FUNCTION_BLOCK FB_Sealer EXTENDS FB_PackML_BaseModule
VAR
    // Sub module definitions here

    // List of sub modules
    ipSubModules_Init : ARRAY[1..Parameters_PackML_Base.MAX_NO_OF_SUBMODULES] OF I_PackML_BaseModule := [];

    // Component definitions here
    SealerAxis : FB_Component_BasicAxis := (Name := 'Axis');
    SealBar    : FB_SealBar             := (Name := 'Heat Bar');

    //Alarms for this module
    SealerAlarms : ARRAY[1..SEALER_ALARM_COUNT] OF FB_TcAlarm;

    //Data for recipe
    Recipe : ST_SealerRecipe;

    (*//Parameters from PackTags for module
    _Param  : ARRAY[1..10] OF ST_Descriptor2;*)
    _Report : ARRAY[1..10] OF ST_Descriptor2;

    //HMI Control for EM
    fbControlSourceHMI : FB_ControlSource_HMI;
END_VAR

VAR CONSTANT

    // Report parameters 
    FAULTID  : INT := 1; //Fault number 
    CURRTEMP : INT := 2; // current temperature of the sealing bar 
    CURRPOS  : INT := 3; // current position of the sealing bar  

    //Alarms
    SEALER_ALARM_COUNT : INT := 6;
END_VAR

//Simulation variables for messaging
VAR
    ErrorInput      : BOOL;
    WarnInput       : BOOL;
    InfoInput       : BOOL;
    TempFeedbackBad : BOOL;
END_VAR

METHOD PROTECTED Aborting
VAR_INPUT
END_VAR
CASE SequenceState OF
    0:
        NoStateTasksToComplete := FALSE;
        SequenceState          := SequenceState + 10;
    10:
        SealBar.Heat := FALSE;
        SealerAxis.Stop();
        IF SealerAxis.Stopped THEN
            SequenceState := SequenceState + 10;
        END_IF
    20:
        // Disable here
        SealerAxis.Disable();

        // Check not enabled here
        IF NOT SealerAxis.Enabled THEN
            SequenceState := SequenceState + 10;
        END_IF
    30:
        StateTasksComplete := TRUE;
END_CASE

SUPER^.Aborting();
END_METHOD

PROPERTY Acceleration : LREAL
SET
Recipe.Axis.Acceleration := Acceleration;
END_SET
END_PROPERTY

METHOD PROTECTED Clearing
VAR_INPUT
END_VAR
CASE SequenceState OF
    0:
        NoStateTasksToComplete := FALSE;
        SequenceState          := SequenceState + 10;
    10:
        // Enable here
        SealerAxis.Enable();

        // Check enabled here
        IF SealerAxis.Enabled THEN
            SequenceState := SequenceState + 10;
        END_IF
    20:
        StateTasksComplete := TRUE;
END_CASE

SUPER^.Clearing();
END_METHOD

PROPERTY ClosedPos : LREAL
GET
ClosedPos := Recipe.ClosedPosition;
END_GET
SET
Recipe.ClosedPosition := ClosedPos;
END_SET
END_PROPERTY

METHOD PROTECTED CreateEvents
VAR_INPUT
END_VAR
// Add your event creation here
F_CreateAllEventsInClass(Alarms     := SealerAlarms,
                         ClassSize  := SIZEOF(TC_EVENTS.Sealer),
                         pInitEvent := ADR(TC_EVENTS.Sealer.InitReferenceEvent),
                         Prefix     := Name);

// Super call to base
SUPER^.CreateEvents();
END_METHOD

METHOD CyclicLogic
VAR_INPUT
END_VAR

VAR
    LowLimit  : STRING;
    HighLimit : STRING;
END_VAR
IF NOT _InitComplete THEN
    _InitComplete := Initialize();
    RETURN;
END_IF

SUPER^.CyclicLogic();
CyclicLogic_Simulation();

//HMI control for EM
fbControlSourceHMI.CyclicLogic();

//Set the current alarm severity for this module
_CurrentAlarmSeverity   := F_GetMaxSeverityRaised(Alarms := SealerAlarms, CurrentSeverity := _CurrentAlarmSeverity);
_Report[CURRTEMP].Value := SealBar.ActualTemperature;
_Report[CURRPOS].Value  := SealerAxis.ActualPosition;

//Monitor seal bar temp
IF NOT SealBar.InTempRange AND NOT SealerAlarms[E_Sealer.TemeratureOutOfRange].bRaised THEN
    LowLimit  := TO_STRING(SealBar.SetTemperature - 1);
    HighLimit := TO_STRING(SealBar.SetTemperature + 1);
    RaiseAlarm2Args(SealerAlarms[E_Sealer.TemeratureOutOfRange], LowLimit, HighLimit);
ELSIF SealBar.InTempRange AND SealerAlarms[E_Sealer.TemeratureOutOfRange].bRaised THEN
    SealerAlarms[E_Sealer.TemeratureOutOfRange].Clear(0, 0);
END_IF
END_METHOD

METHOD CyclicLogic_Simulation
VAR_INPUT
END_VAR

VAR_INST
END_VAR
(*	
This is just for testing. Real hardware can be setup in other places
Here the alarms will raise and clear on its own if the input changes	
*)

//Generic Alarms for Testing
IF ErrorInput AND NOT SealerAlarms[E_Sealer.AlarmMessage].bRaised THEN
    RaiseAlarm2Args(SealerAlarms[E_Sealer.AlarmMessage], '', '');
ELSIF NOT ErrorInput AND SealerAlarms[E_Sealer.AlarmMessage].bRaised THEN
    SealerAlarms[E_Sealer.AlarmMessage].Clear(0, 0);
END_IF

IF WarnInput AND NOT SealerAlarms[E_Sealer.WarnMessage].bRaised THEN
    RaiseAlarm2Args(SealerAlarms[E_Sealer.WarnMessage], '', '');
ELSIF NOT WarnInput AND SealerAlarms[E_Sealer.WarnMessage].bRaised THEN
    SealerAlarms[E_Sealer.WarnMessage].Clear(0, 0);
END_IF

IF InfoInput AND NOT SealerAlarms[E_Sealer.InfoMessage].bRaised THEN
    RaiseAlarm2Args(SealerAlarms[E_Sealer.InfoMessage], '', '');
ELSIF NOT InfoInput AND SealerAlarms[E_Sealer.InfoMessage].bRaised THEN
    SealerAlarms[E_Sealer.InfoMessage].Clear(0, 0);
END_IF

// Only here for simulating alarm
IF TempFeedbackBad AND NOT SealerAlarms[E_Sealer.FeedbackError].bRaised THEN
    RaiseAlarm2Args(SealerAlarms[E_Sealer.FeedbackError], '', '');
ELSIF NOT TempFeedbackBad AND SealerAlarms[E_Sealer.FeedbackError].bRaised THEN
    SealerAlarms[E_Sealer.FeedbackError].Clear(0, 0);
END_IF
END_METHOD

METHOD PROTECTED Execute
VAR_INPUT
END_VAR

VAR_INST
    dwellTime : TON;
END_VAR
CASE _CurrentMode OF
    //=================================PRODUCTION MODE==================================
    E_PMLUnitMode.ePMLUnitMode_Production:
        CASE SequenceState OF
            0:
                IF SealerAxis.InPosition AND NOT SealerAxis.Busy THEN
                    /// SealerAxis needs to do reporting here?? no tags in the components for PackML so should be done with this module
                    dwellTime(IN := TRUE, PT := LREAL_TO_TIME(Recipe.SealTime));
                    SequenceState := SequenceState + 10;
                END_IF
            10:
                IF dwellTime.Q THEN
                    dwellTime(IN := FALSE);
                    SealerAxis.Velocity     := Recipe.Axis.Velocity;    
                    SealerAxis.Acceleration := Recipe.Axis.Acceleration;
                    SealerAxis.MoveAbsolute(Position := Recipe.OpenPosition, FALSE);
                    SequenceState := SequenceState + 10;
                END_IF
            20:
                IF SealerAxis.InPosition AND NOT SealerAxis.Busy THEN
                    ///SealerAxis report position?
                    StateComplete();
                END_IF
        END_CASE

        dwellTime();

    //=================================MAINTENANCE & MANUAL MODE==================================		
    E_PMLUnitMode.ePMLUnitMode_Maintenance, E_PMLUnitMode.ePMLUnitMode_Manual:
        ;
END_CASE
END_METHOD

PROPERTY Heat : BOOL
GET
Heat := SealBar.Heat;
END_GET
SET
SealBar.Heat := Heat;
END_SET
END_PROPERTY

//! @summary Basic module initialization logic
METHOD PROTECTED Initialize : BOOL;
VAR
    i                        : UDINT;
    varInfo                  : __SYSTEM.VAR_INFO;
    AllSubUnitsInitialized   : BOOL := TRUE;
    AllComponentsInitialized : BOOL := TRUE;
END_VAR

//! @description This method is called by <c>CyclicLogic()</c> as required
Initialize := FALSE;
CASE DescendantSequenceState OF
    0:
		RegisterComponent(SealerAxis);
		RegisterComponent(SealBar);
		
        _LogModeChanges         := FALSE;
        _LogStateChanges        := FALSE;
        DescendantSequenceState := DescendantSequenceState + 10;
    10:
        //Setup Custom modes here

        (*CustomModes(eMode                          :=,
                    sName                          :=,
                    bDisableClearing               :=,
                    bDisableStarting               :=,
                    bDisableSuspended              :=,
                    bDisableStopping               :=,
                    bDisableAborting               :=,
                    bDisableHolding                :=,
                    bDisableHeld                   :=,
                    bDisableUnholding              :=,
                    bDisableSuspending             :=,
                    bDisableUnsuspending           :=,
                    bDisableResetting              :=,
                    bDisableIdle                   :=,
                    bDisableCompleting             :=,
                    bDisableComplete               :=,
                    bEnableUnitModeChangeStopped   :=,
                    bEnableUnitModeChangeIdle      :=,
                    bEnableUnitModeChangeSuspended :=,
                    bEnableUnitModeChangeExecute   :=,
                    bEnableUnitModeChangeAborted   :=,
                    bEnableUnitModeChangeHeld      :=,
                    bEnableUnitModeChangeComplete  :=,
                    bError                         =>,
                    nErrorId                       =>);*)
        DescendantSequenceState := DescendantSequenceState + 10;
    20:
        //Copy Mode names
        FOR i := 1 TO 3 DO
            ModeNames[i] := F_UnitModeToString(UDINT_TO_DINT(i));
        END_FOR

        Initialize_TagData();
		RegisterExternalController(Controller := fbControlSourceHMI);
		fbControlSourceHMI.CyclicLogic();
        DescendantSequenceState := DescendantSequenceState + 10;
    30:
        //Call the Super
        IF SUPER^.Initialize() THEN
            DescendantSequenceState := DescendantSequenceState + 10;
        END_IF
    40:
        Initialize := TRUE;
END_CASE
END_METHOD

METHOD Initialize_TagData
VAR_INPUT
END_VAR
//Reports
_Report[FAULTID].ID    := TO_DINT(2 * 10 + 1);
_Report[FAULTID].Name  := 'Fault';
_Report[FAULTID].Unit  := '';
_Report[CURRPOS].ID    := TO_DINT(2 * 10 + 2);
_Report[CURRPOS].Name  := 'Seal Pos';
_Report[CURRPOS].Unit  := 'deg';
_Report[CURRTEMP].ID   := TO_DINT(2 * 10 + 3);
_Report[CURRTEMP].Name := 'Seal Temp';
_Report[CURRTEMP].Unit := 'C';

// Recipe
Recipe.Axis.Velocity     := 100;
Recipe.Axis.Acceleration := 1000;
Recipe.ClosedPosition    := 200;
Recipe.OpenPosition      := 105;
Recipe.Temp              := 100;
Recipe.SealTime          := 250;
END_METHOD

PROPERTY OpenPos : LREAL
GET
OpenPos := Recipe.OpenPosition;
END_GET
SET
Recipe.OpenPosition := OpenPos;
END_SET
END_PROPERTY

METHOD RaiseAlarm2Args
VAR_IN_OUT
    Alarm : FB_TcAlarm; //Alarm to be raised
END_VAR

VAR_INPUT
    String_1 : STRING; //First String Parameter (The Name of this component will be applied first automatically)
    String_2 : STRING; //Second String Parameter
END_VAR
F_RaiseAlarmWithStringParameters(Alarm    := Alarm,
                                 String_1 := Name,
                                 String_2 := String_1,
                                 String_3 := String_2);
END_METHOD

PROPERTY SealTime : LREAL
GET
SealTime := Recipe.SealTime;
END_GET
SET
Recipe.SealTime := SealTime;
END_SET
END_PROPERTY

METHOD PROTECTED Starting
VAR_INPUT
END_VAR
CASE _CurrentMode OF
    //=================================PRODUCTION MODE==================================
    E_PMLUnitMode.ePMLUnitMode_Production:
        CASE SequenceState OF
            0:
                NoStateTasksToComplete := FALSE;
                SequenceState          := SequenceState + 10;
            10:
                SealerAxis.Velocity     := Recipe.Axis.Velocity;
                SealerAxis.Acceleration := Recipe.Axis.Acceleration;
                SealerAxis.MoveAbsolute(Position := Recipe.ClosedPosition, FALSE);
                SequenceState := SequenceState + 10;
            20:
                IF SealerAxis.Busy THEN
                    StateTasksComplete := TRUE;
                END_IF
        END_CASE

    //=================================MAINTENANCE & MANUAL MODE==================================
    E_PMLUnitMode.ePMLUnitMode_Maintenance, E_PMLUnitMode.ePMLUnitMode_Manual:
        ;
END_CASE

SUPER^.Starting();
END_METHOD

PROPERTY Temp : LREAL
GET
Temp := Recipe.Temp;
END_GET
SET
Recipe.Temp := Temp;
SealBar.SetTemperature := Recipe.Temp;
END_SET
END_PROPERTY

PROPERTY Velocity : LREAL
SET
Recipe.Axis.Velocity := Velocity;
END_SET
END_PROPERTY

END_FUNCTION_BLOCK

(* stored: Version 1.1.0.1
   POU FB_Sealer: Id {ff58966f-3da2-41b5-b2fb-39a4520ba938}, SpecialFunc None
   Folder I_CyclicFB: Id {2bf8202d-347a-4b96-8511-350b7ced3b49}
   Folder Methods: Id {87e89e76-36f1-4ae7-ab6f-dd985ead3154}
   Folder Acting States: Id {83c2fb32-603a-4bf1-b0d3-b82fdb72188e}
   Folder WaitingStates: Id {c5fb234c-f50f-4161-be0e-18f57c35714d}
   Folder Properties: Id {f36d5a6c-14e3-49a8-bae7-9fd37d1c0349}
   Method Aborting: Id {b6180b57-df4e-43ee-a76d-c9274b8854f0}
   Property Acceleration: Id {daa0dee7-a9eb-47e2-99ea-3fb9b5a6407e}
   Set Set: Id {c26780f0-3bf0-41e2-a963-3d1b2ba97499}
   Method Clearing: Id {15caa36d-4f9c-40b9-b52a-3d58374eb0b3}
   Property ClosedPos: Id {68701d47-5346-4cb2-9de1-742627e7e729}
   Get Get: Id {c06b5f0b-e909-4d36-88d6-121b089c55f9}
   Set Set: Id {efc7f76a-0a9f-4b42-b34b-b37c43fadacc}
   Method CreateEvents: Id {6e6ca775-6d05-4f9d-acb6-719514de2f41}
   Method CyclicLogic: Id {556f07f6-dd73-4758-81e0-ff19676cbbed}
   Method CyclicLogic_Simulation: Id {cb7b038b-49dc-4f4e-b388-330c9a9651b1}
   Method Execute: Id {e9b1fd0e-8980-4f06-b93a-7f213fd426be}
   Property Heat: Id {3bbb6d28-e767-45db-b8a5-70445d97c848}
   Get Get: Id {46a2d081-1dab-4ce7-8b6f-978d995de8e1}
   Set Set: Id {e760ac7c-03a2-4cd5-a5f2-c5dad5acc2b4}
   Method Initialize: Id {46d90c83-0de6-49f0-8e5c-f5f7ebdc808d}
   Method Initialize_TagData: Id {ca3d7819-a229-4f43-b3dc-1b676f338712}
   Property OpenPos: Id {f80892fd-0de7-4951-a1c3-9a2675bea75d}
   Get Get: Id {cc65af72-d546-43b6-8e91-4313a8c1faff}
   Set Set: Id {c927aad9-2e51-4c56-bacc-1e989b479fa0}
   Method RaiseAlarm2Args: Id {50d20dd4-a4f9-4638-962e-3d6308ad4688}
   Property SealTime: Id {9e06eaf2-efc2-4fc7-bea7-d2c9244a59b5}
   Get Get: Id {012f31e5-11ae-4a29-93bb-9fb67f60939c}
   Set Set: Id {5f0e1a8f-33da-416f-b952-1dddfa44d7e0}
   Method Starting: Id {d8069b32-aac5-4160-8750-2cb4e87a420f}
   Property Temp: Id {75cb2623-9ee1-491d-a300-c94bd0c0a581}
   Get Get: Id {60c0dab2-2395-4335-80da-14e31abceed6}
   Set Set: Id {fea897ac-3069-449a-926e-882752ac4fa8}
   Property Velocity: Id {82c39321-7609-4946-b7fc-d3898485c4c7}
   Set Set: Id {c6fdb1c6-b663-4277-b18d-e2c9a4196149} *)
